PROGRAM MAIN
VAR
END_VAR

END_PROGRAM

(* stored: Version 1.1.0.1
   POU MAIN: Id {bd45a85e-c83e-4a53-bc0e-3b956a609f08} *)
